SUBAPPLICATION TageszaehlerVergleich (* Subapplication Type *)
  (* Standard: 61499-2 *)
  (* Version 1.0, 2023-02-18, Franz *)
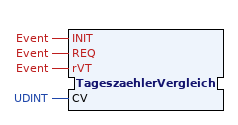
  EVENT_INPUT
    INIT; (* Initialization Request *)
    REQ; (* Normal Execution Request *)
    rVT; (* refresh VT *)
  END_EVENT
  VAR_INPUT
    CV : UDINT; (* Counter Value *)
  END_VAR
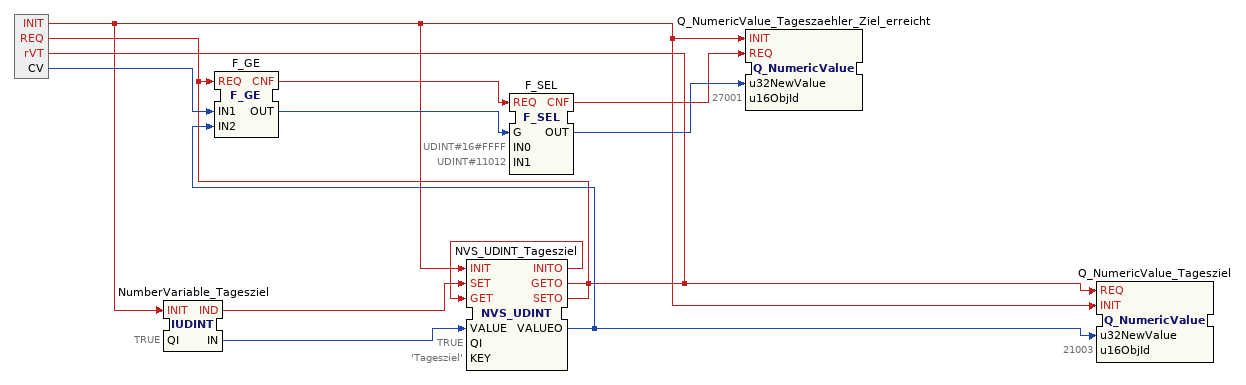
  FBS
    Q_NumericValue_Tageszaehler_Ziel_erreicht : Q_NumericValue(u16ObjId := 27001);
    F_GE : F_GE;
    F_SEL : F_SEL(IN0 := UDINT#16#FFFF, IN1 := UDINT#11012);
    NVS_UDINT_Tagesziel : NVS_UDINT(QI := TRUE, KEY := 'Tagesziel');
    NumberVariable_Tagesziel : IUDINT(QI := TRUE);
    Q_NumericValue_Tagesziel : Q_NumericValue(u16ObjId := 21003);
  END_FBS
  EVENT_CONNECTIONS
    INIT TO Q_NumericValue_Tageszaehler_Ziel_erreicht.INIT;
    REQ TO F_GE.REQ;
    F_GE.CNF TO F_SEL.REQ;
    F_SEL.CNF TO Q_NumericValue_Tageszaehler_Ziel_erreicht.REQ;
    INIT TO NumberVariable_Tagesziel.INIT;
    INIT TO NVS_UDINT_Tagesziel.INIT;
    NumberVariable_Tagesziel.IND TO NVS_UDINT_Tagesziel.SET;
    NVS_UDINT_Tagesziel.INITO TO NVS_UDINT_Tagesziel.GET;
    NVS_UDINT_Tagesziel.GETO TO Q_NumericValue_Tagesziel.REQ;
    INIT TO Q_NumericValue_Tagesziel.INIT;
    NVS_UDINT_Tagesziel.GETO TO F_GE.REQ;
    NVS_UDINT_Tagesziel.SETO TO F_GE.REQ;
    rVT TO Q_NumericValue_Tagesziel.REQ;
  END_CONNECTIONS
  DATA_CONNECTIONS
    CV TO F_GE.IN1;
    F_SEL.OUT TO Q_NumericValue_Tageszaehler_Ziel_erreicht.u32NewValue;
    F_GE.OUT TO F_SEL.G;
    NumberVariable_Tagesziel.IN TO NVS_UDINT_Tagesziel.VALUE;
    NVS_UDINT_Tagesziel.VALUEO TO Q_NumericValue_Tagesziel.u32NewValue;
    NVS_UDINT_Tagesziel.VALUEO TO F_GE.IN2;
  END_CONNECTIONS
END_SUBAPPLICATION
